// TIA Portal V17 export
// export: Created 2023-12-22T15:05:34.1947016Z, ExportSetting WithDefaults, DisplayName Totally Integrated Automation Portal, DisplayVersion V17, DisplayName TIA Portal Openness, DisplayVersion V17, DisplayName TIA Portal Version Control Interface, DisplayVersion V17, DisplayName STEP 7 Professional, DisplayVersion V17, DisplayName STEP 7 Safety, DisplayVersion V17, DisplayName WinCC Advanced, DisplayVersion V17
DATA_BLOCK "Line_Control_DB"   // DB5
VERSION : 0.1
// stored: AutoNumber false, DBAccessibleFromOPCUA true, InstanceOfName Line_Control, InstanceOfType FB
"Line_Control"
   // VAR RETAIN
   //    Local : Bool;
   //    RESET_STAT : Bool;
   //    Line_Settings : Bool;
   //    Line_Alarms : Bool;
   //    Group1_PolyMix_1 : Bool;
   //    Group1_PolyMix_2 : Bool;
   //    Group2_PolyMix_1 : Bool;
   //    Group2_PolyMix_2 : Bool;
   //    ALLS : Bool;
   //    REQ_Z6_BK1 : Bool;
   //    REQ_Z6_BK2 : Bool;
   //    REQ_Z5_Start_A : Bool;
   //    REQ_Z4_Start_A : Bool;
   //    REQ_Z3_Start_A : Bool;
   //    REQ_Z2_Start_A : Bool;
   //    REQ_Z1_Start_A : Bool;
   //    Line_REQ_Settings : Int;
   //    Line_Now_Settings : Int;
   //    Line_REQ_Alarms : Int;
   //    Line_Now_Alarms : Int;
   //    All_Lines : Int := 2;
   //    All_Pumps : Int := 2;
   //    Events : Word;
   //    pos : Array[0..7] of Bool;
   //    Line { S7_SetPoint := 'True'} : Array[0..2] of "Block_Line";
   //    Pump { S7_SetPoint := 'True'} : Array[1..2] of "Block_Pump";
   //    Time_DTL : DTL;
   // END_VAR
BEGIN
   Line[0..2].Hand := FALSE;
   Line[0..2].SP_Source := TRUE;
   Line[0..2].PID_Not_Use := FALSE;
   Line[0..2].Mode := FALSE;
   Line[0..2].RM_1_Report_DI := FALSE;
   Line[0..2].RM_2_Report_DI := FALSE;
   Line[0..2].RM_Weight := 1.0;
   Line[0].SP_M := 0.0;
   Line[1].SP_M := 1.0;
   Line[2].SP_M := 0.0;
   Line[0..2].SP_min := 10.0;
   Line[0..2].SP_max := 200.0;
   Line[0..2].PE_min := 0.15;
   Line[0..2].PE_max := 2.5;
   Line[0..2].D := 0.0;
   Line[0..2].C_Tank := 0.0;
   Line[0..2].Low_Flow := 0.0;
   Line[0].Res_SP := 0.0;
   Line[1].Res_SP := 4.0;
   Line[2].Res_SP := 0.0;
   Line[0..2].Use.RT := FALSE;
   Line[0..2].Use.RM := FALSE;
   Line[0..2].Use.SP := TRUE;
   Line[0..2].Use.Flow := FALSE;
   Line[0..2].Use.Res := FALSE;
   Line[0..2].Use.DME := FALSE;
   Line[0..2].Use.PE := FALSE;
   Line[0..2].PID.CMD.Vector := FALSE;
   Line[0..2].PID.x := 1.0;
   Line[0..2].PID.Settings.SP_P := 1.5;
   Line[0..2].PID.Settings.SP_Ti := 150.0;
   Line[0..2].PID.Settings.SP_Td := 0.0;
   Line[0..2].PID.Settings.SP_Cycle := 0.2;
   Line[0..2].PID.Settings.Max_SP := 500.0;
   Line[0..2].PID.Settings.Min_SP := -500.0;
   Line[0..2].PID.Settings.Max_in := 500.0;
   Line[0..2].PID.Settings.Min_in := -500.0;
   Line[0..2].PID.Settings.Max_out := 100.0;
   Line[0..2].PID.Settings.Min_out := 0.0;
   Line[0].PID.Settings.DeadBand := 0.0;
   Line[1..2].PID.Settings.DeadBand := 1.0;
   Line[0..2].PID.PID.IntegralResetMode := 4;
   Line[0..2].PID.PID.RunModeByStartup := TRUE;
   Line[0..2].PID.PID.SetSubstituteOutput := TRUE;
   Line[0..2].PID.PID.ActivateRecoverMode := TRUE;
   Line[0..2].PID.PID.CancelTuningLevel := 10.0;
   Line[0..2].PID.PID.SubstituteOutput := 0.0;
   Line[0].PID.PID.Config.InputPerOn := TRUE;
   Line[1..2].PID.PID.Config.InputPerOn := FALSE;
   Line[0..2].PID.PID.Config.InvertControl := FALSE;
   Line[0].PID.PID.Config.InputUpperLimit := 120.0;
   Line[1..2].PID.PID.Config.InputUpperLimit := 500.0;
   Line[0].PID.PID.Config.InputLowerLimit := 0.0;
   Line[1..2].PID.PID.Config.InputLowerLimit := -500.0;
   Line[0..2].PID.PID.Config.InputUpperWarning := 3.402822E+38;
   Line[0..2].PID.PID.Config.InputLowerWarning := -3.402822E+38;
   Line[0..2].PID.PID.Config.OutputUpperLimit := 100.0;
   Line[0..2].PID.PID.Config.OutputLowerLimit := 0.0;
   Line[0].PID.PID.Config.SetpointUpperLimit := 3.402822E+38;
   Line[1..2].PID.PID.Config.SetpointUpperLimit := 500.0;
   Line[0].PID.PID.Config.SetpointLowerLimit := -3.402822E+38;
   Line[1..2].PID.PID.Config.SetpointLowerLimit := -500.0;
   Line[0..2].PID.PID.Config.MinimumOnTime := 0.0;
   Line[0..2].PID.PID.Config.MinimumOffTime := 0.0;
   Line[0..2].PID.PID.Config.InputScaling.UpperPointIn := 27648.0;
   Line[0..2].PID.PID.Config.InputScaling.LowerPointIn := 0.0;
   Line[0..2].PID.PID.Config.InputScaling.UpperPointOut := 100.0;
   Line[0..2].PID.PID.Config.InputScaling.LowerPointOut := 0.0;
   Line[0..2].PID.PID.CycleTime.EnEstimation := TRUE;
   Line[0..2].PID.PID.CycleTime.EnMonitoring := TRUE;
   Line[0].PID.PID.CycleTime.Value := 0.1;
   Line[1].PID.PID.CycleTime.Value := 0.2005259;
   Line[2].PID.PID.CycleTime.Value := 0.2005263;
   Line[0..2].PID.PID.CtrlParamsBackUp.Gain := 1.0;
   Line[0..2].PID.PID.CtrlParamsBackUp.Ti := 20.0;
   Line[0..2].PID.PID.CtrlParamsBackUp.Td := 0.0;
   Line[0..2].PID.PID.CtrlParamsBackUp.TdFiltRatio := 0.2;
   Line[0..2].PID.PID.CtrlParamsBackUp.PWeighting := 1.0;
   Line[0..2].PID.PID.CtrlParamsBackUp.DWeighting := 1.0;
   Line[0..2].PID.PID.CtrlParamsBackUp.Cycle := 1.0;
   Line[0].PID.PID.PIDSelfTune.SUT.TuneRule := 0;
   Line[1..2].PID.PID.PIDSelfTune.SUT.TuneRule := 1;
   Line[0..2].PID.PID.PIDSelfTune.TIR.TuneRule := 0;
   Line[0].PID.PID.Retain.CtrlParams.Gain := 1.0;
   Line[1..2].PID.PID.Retain.CtrlParams.Gain := 1.5;
   Line[0].PID.PID.Retain.CtrlParams.Ti := 20.0;
   Line[1..2].PID.PID.Retain.CtrlParams.Ti := 150.0;
   Line[0..2].PID.PID.Retain.CtrlParams.Td := 0.0;
   Line[0..2].PID.PID.Retain.CtrlParams.TdFiltRatio := 0.2;
   Line[0..2].PID.PID.Retain.CtrlParams.PWeighting := 1.0;
   Line[0..2].PID.PID.Retain.CtrlParams.DWeighting := 1.0;
   Line[0..2].PID.PID.Retain.CtrlParams.Cycle := 1.0;
   Line[0].PID.C.SP := 1.0;
   Line[1..2].PID.C.SP := 0.2;
   Line[0..2].PID.C.One := 0.1;
   Line[0].FlowMeter_1.Mode := FALSE;
   Line[1..2].FlowMeter_1.Mode := TRUE;
   Line[0..2].FlowMeter_1.Fast_Mode := TRUE;
   Line[0..2].FlowMeter_1.clock := 0.01;
   Line[0..2].FlowMeter_1.Weight := 1.0;
   Line[0..2].FlowMeter_1.All := 0.0;
   Line[0..2].FlowMeter_1.Any := 0.0;
   Line[0..2].FlowMeter_1.Seans := 0.0;
   Line[0..2].FlowMeter_1.Seans_Last := 0.0;
   Line[0].FlowMeter_1.Flow_Today := 0.0;
   Line[1..2].FlowMeter_1.Flow_Today := 0.3833334;
   Line[0].FlowMeter_1.Flow_LastDay := 0.0;
   Line[1].FlowMeter_1.Flow_LastDay := 0.3833334;
   Line[2].FlowMeter_1.Flow_LastDay := 0.0;
   Line[0..2].FlowMeter_1.Flow_Lock_All := 0.0;
   Line[0..2].FlowMeter_1.Flow_Lock_Now := 0.0;
   Line[0].FlowMeter_1.ADDR_Byte := 0;
   Line[1].FlowMeter_1.ADDR_Byte := 2;
   Line[2].FlowMeter_1.ADDR_Byte := 0;
   Line[0].FlowMeter_1.ADDR_Bit := 0;
   Line[1].FlowMeter_1.ADDR_Bit := 1;
   Line[2].FlowMeter_1.ADDR_Bit := 0;
   Line[0..2].FlowMeter_1.Filter.Moment := TRUE;
   Line[0].FlowMeter_2.Mode := FALSE;
   Line[1..2].FlowMeter_2.Mode := TRUE;
   Line[0..2].FlowMeter_2.Fast_Mode := TRUE;
   Line[0..2].FlowMeter_2.clock := 0.01;
   Line[0..2].FlowMeter_2.Weight := 1.0;
   Line[0..2].FlowMeter_2.All := 0.0;
   Line[0..2].FlowMeter_2.Any := 0.0;
   Line[0..2].FlowMeter_2.Seans := 0.0;
   Line[0..2].FlowMeter_2.Seans_Last := 0.0;
   Line[0..2].FlowMeter_2.Flow_Today := 0.0;
   Line[0..2].FlowMeter_2.Flow_LastDay := 0.0;
   Line[0..2].FlowMeter_2.Flow_Lock_All := 0.0;
   Line[0..2].FlowMeter_2.Flow_Lock_Now := 0.0;
   Line[0..2].FlowMeter_2.ADDR_Byte := 0;
   Line[0..2].FlowMeter_2.ADDR_Bit := 0;
   Line[0..2].FlowMeter_2.Filter.Moment := TRUE;
   Pump[1..2].Reserv := FALSE;
   Pump[1..2].Line_Main := 1;
   Pump[1..2].Line_Reserv := 0;
END_DATA_BLOCK
